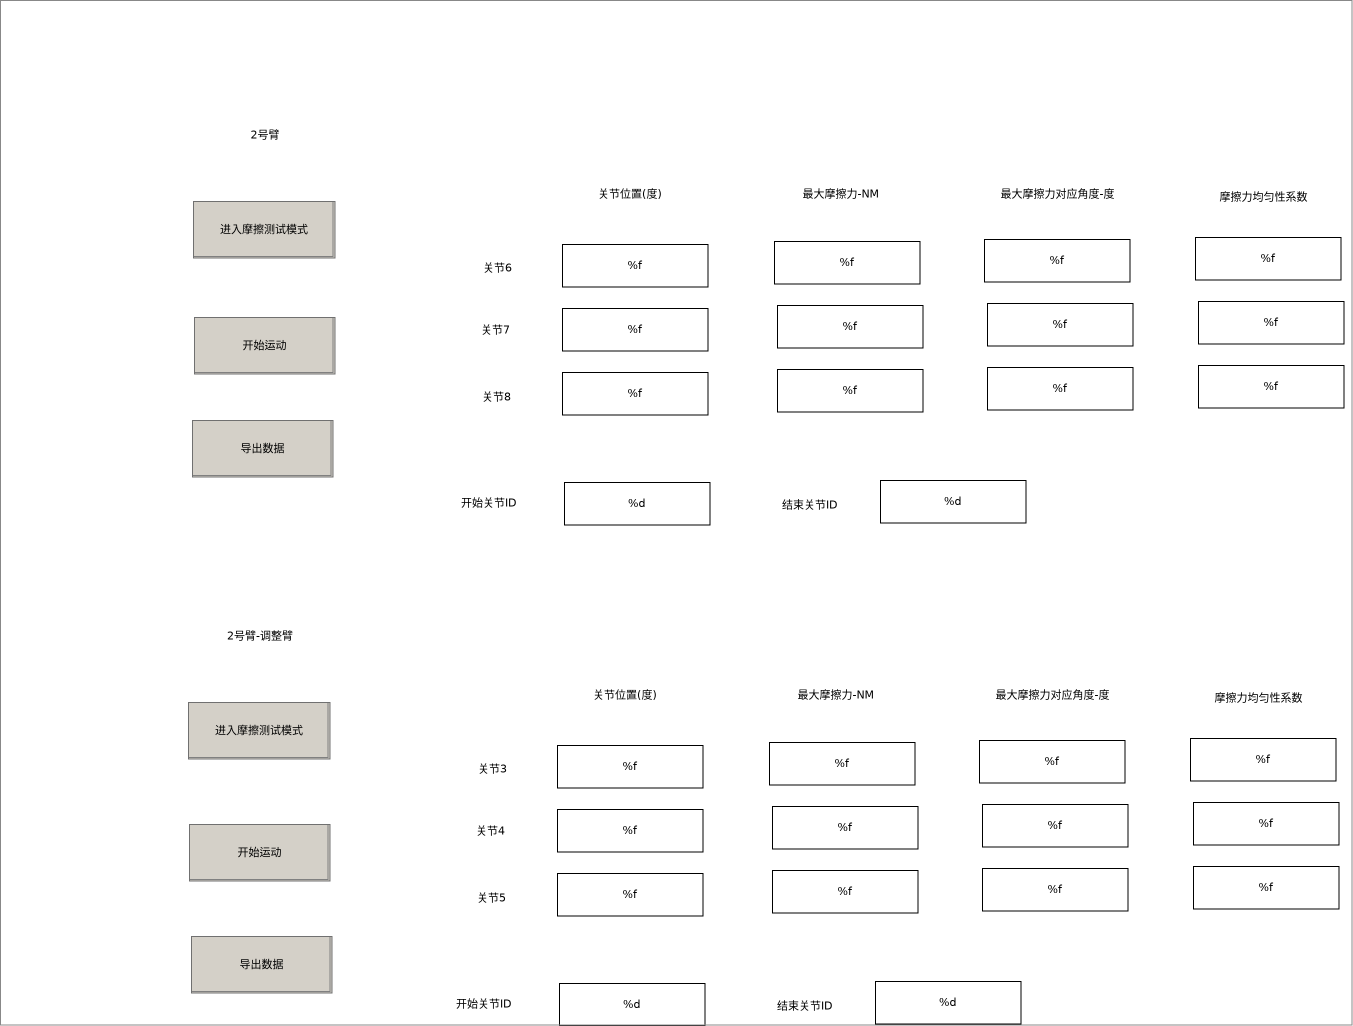
VISUALIZATION friction_a2  // 1353x1026
    Button (193,201 142x57), "进入摩擦测试模式", colour toggle: g_frictionTest.m_testMode[2]
        toggle g_frictionTest.m_testMode[2]
    Button (194,317 141x57), "开始运动", colour toggle: g_frictionTest.m_startMotion[2]
        toggle g_frictionTest.m_startMotion[2]
    Label (190,120 150x30), "2号臂"
    Rectangle (774,241 146x43), "%f", text variable: g_frictionTest.m_CoulombFrictionMax[2][1]
    Rectangle (777,305 146x43), "%f", text variable: g_frictionTest.m_CoulombFrictionMax[2][2]
    Rectangle (777,369 146x43), "%f", text variable: g_frictionTest.m_CoulombFrictionMax[2][3]
    Label (766,179 150x30), "最大摩擦力-NM"
    Rectangle (984,239 146x43), "%f", text variable: g_frictionTest.m_CoulombFrictionMax_JntPos[2][1]
    Rectangle (987,303 146x43), "%f", text variable: g_frictionTest.m_CoulombFrictionMax_JntPos[2][2]
    Rectangle (987,367 146x43), "%f", text variable: g_frictionTest.m_CoulombFrictionMax_JntPos[2][3]
    Label (941,179 233x30), "最大摩擦力对应角度-度"
    Rectangle (1195,237 146x43), "%f", text variable: g_frictionTest.m_CoulombFrictionRatio[2,1]
    Rectangle (1198,301 146x43), "%f", text variable: g_frictionTest.m_CoulombFrictionRatio[2,2]
    Rectangle (1198,365 146x43), "%f", text variable: g_frictionTest.m_CoulombFrictionRatio[2,3]
    Label (1174,182 179x30), "摩擦力均匀性系数"
    Rectangle (562,244 146x43), "%f", text variable: g_frictionTest.m_armDHJntPos[2][1]
    Label (446,250 103x36), "关节6"
    Label (444,312 103x36), "关节7"
    Label (445,379 103x36), "关节8"
    Rectangle (562,308 146x43), "%f", text variable: g_frictionTest.m_armDHJntPos[2][2]
    Rectangle (562,372 146x43), "%f", text variable: g_frictionTest.m_armDHJntPos[2][3]
    Label (555,179 150x30), "关节位置(度)"
    Label (414,488 150x30), "开始关节ID"
    Rectangle (564,482 146x43), "%d", text variable: g_frictionTest.m_jntIdStart[2]
        OnMouseClick: write the text variable via Default
    Label (735,490 150x30), "结束关节ID"
    Rectangle (880,480 146x43), "%d", text variable: g_frictionTest.m_jntIdEnd[2]
        OnMouseClick: write the text variable via Default
    Button (188,702 142x57), "进入摩擦测试模式", colour toggle: g_frictionTestSetup.m_testMode[2]
        toggle g_frictionTestSetup.m_testMode[2]
    Button (189,824 141x57), "开始运动", colour toggle: g_frictionTestSetup.m_startMotion[2]
        toggle g_frictionTestSetup.m_startMotion[2]
    Label (185,621 150x30), "2号臂-调整臂"
    Rectangle (769,742 146x43), "%f", text variable: g_frictionTestSetup.m_CoulombFrictionMax[2][3]
    Rectangle (772,806 146x43), "%f", text variable: g_frictionTestSetup.m_CoulombFrictionMax[2][4]
    Rectangle (772,870 146x43), "%f", text variable: g_frictionTestSetup.m_CoulombFrictionMax[2][5]
    Label (761,680 150x30), "最大摩擦力-NM"
    Rectangle (979,740 146x43), "%f", text variable: g_frictionTestSetup.m_CoulombFrictionMax_JntPos[2][3]
    Rectangle (982,804 146x43), "%f", text variable: g_frictionTestSetup.m_CoulombFrictionMax_JntPos[2][4]
    Rectangle (982,868 146x43), "%f", text variable: g_frictionTestSetup.m_CoulombFrictionMax_JntPos[2][5]
    Label (936,680 233x30), "最大摩擦力对应角度-度"
    Rectangle (1190,738 146x43), "%f", text variable: g_frictionTestSetup.m_CoulombFrictionRatio[2,3]
    Rectangle (1193,802 146x43), "%f", text variable: g_frictionTestSetup.m_CoulombFrictionRatio[2,4]
    Rectangle (1193,866 146x43), "%f", text variable: g_frictionTestSetup.m_CoulombFrictionRatio[2,5]
    Label (1169,683 179x30), "摩擦力均匀性系数"
    Rectangle (557,745 146x43), "%f", text variable: g_frictionTestSetup.m_armDHJntPos[2][3]
    Label (441,751 103x36), "关节3"
    Label (439,813 103x36), "关节4"
    Label (440,880 103x36), "关节5"
    Rectangle (557,809 146x43), "%f", text variable: g_frictionTestSetup.m_armDHJntPos[2][4]
    Rectangle (557,873 146x43), "%f", text variable: g_frictionTestSetup.m_armDHJntPos[2][5]
    Label (550,680 150x30), "关节位置(度)"
    Label (409,989 150x30), "开始关节ID"
    Rectangle (559,983 146x43), "%d", text variable: g_frictionTestSetup.m_jntIdStart[2]
        OnMouseClick: write the text variable via Default
    Label (730,991 150x30), "结束关节ID"
    Rectangle (875,981 146x43), "%d", text variable: g_frictionTestSetup.m_jntIdEnd[2]
        OnMouseClick: write the text variable via Default
    Button (192,420 141x57), "导出数据", colour toggle: g_frictionTest.m_duringWriteData[2]
        tap g_frictionTest.m_writeData[2]
    Button (191,936 141x57), "导出数据", colour toggle: g_frictionTestSetup.m_duringWriteData[2]
        tap g_frictionTestSetup.m_writeData[2]
END_VISUALIZATION

(* stored: Version 1.1.0.1, ProductVersion 3.1.4024.11
   Visu friction_a2: Id {c5da6a10-b4de-4783-9cb5-6c5f69b125f7} *)
